ABB RAPID module: tester_right.mod

MODULE tester_right
LOCAL CONST string YuMi_App_Program_Version:="1.0.1"; !Do not edit or remove this line!
LOCAL VAR robtarget s7 := [[511.381,-219.339,941.704],[0.137031,-0.253187,0.090374,-0.953389],[-1,-4,-3,100],[123.501,9E+09,9E+09,9E+09,9E+09,9E+09]];
LOCAL VAR robtarget s6 := [[447.511,-378.152,479.729],[0.0142443,0.564229,-0.79712,0.214575],[-1,-1,0,110],[-45.0976,9E+09,9E+09,9E+09,9E+09,9E+09]];
LOCAL VAR robtarget s5 := [[212.276,-51.1605,1133.79],[0.103913,0.454277,0.298995,0.832728],[-1,0,-1,110],[-27.7686,9E+09,9E+09,9E+09,9E+09,9E+09]];
LOCAL VAR robtarget s4 := [[312.949,-68.6994,1050.79],[0.0696119,0.196396,-0.873676,-0.439627],[-1,1,-2,110],[-22.5579,9E+09,9E+09,9E+09,9E+09,9E+09]];
LOCAL VAR robtarget s3 := [[470.166,-465.155,446.597],[0.606062,-0.370346,0.315644,0.629207],[0,0,1,110],[-27.7693,9E+09,9E+09,9E+09,9E+09,9E+09]];
LOCAL VAR robtarget s2 := [[191.427,-360.211,784.317],[0.380315,0.517245,0.188283,-0.743215],[0,-4,1,1100],[134.5,9E+09,9E+09,9E+09,9E+09,9E+09]];
LOCAL VAR robtarget s1 := [[188.26,-245.486,707.695],[0.444661,0.567091,-0.315644,-0.617295],[0,-4,2,110],[19.1688,9E+09,9E+09,9E+09,9E+09,9E+09]];
PROC main()
MoveSync s1;
MoveSync s2;
MoveSync s3;
MoveSync s4;
MoveSync s5;
MoveSync s6;
MoveSync s7;
ENDPROC
ENDMODULE
